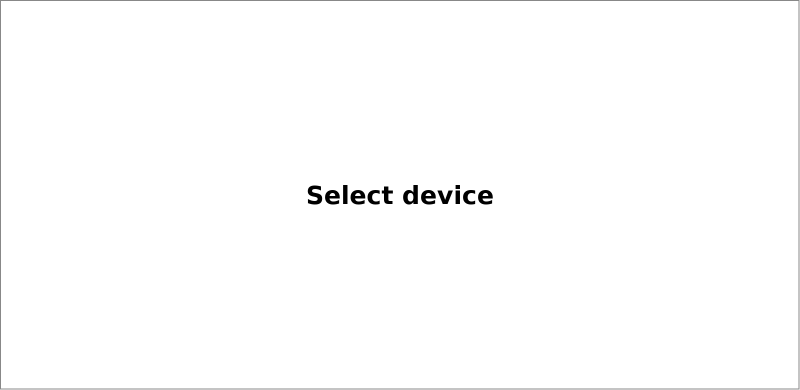
VISUALIZATION VisuUndefinedControl  // 800x390
    Label (0,0 800x390), "Select device"
END_VISUALIZATION

(* stored: Version 1.1.0.1, ProductVersion 3.1.4024.11
   Visu VisuUndefinedControl: Id {aa3a56b2-99b4-0c95-1560-2d5f40cd8538} *)
